// TIA Portal V17 export
// export: Created 2025-03-10T13:11:49.6492455Z, ExportSetting WithDefaults, DisplayName Totally Integrated Automation Portal, DisplayVersion V17 Update 8, DisplayName TIA Portal Openness, DisplayVersion V17 Update 8, DisplayName TIA Portal Version Control Interface, DisplayVersion V17, DisplayName SINAMICS Startdrive Advanced, DisplayVersion V17 SP2, DisplayName SINAMICS Startdrive G110M, G120, G120C, G120D, G120P, G115D, DisplayVersion V17 SP2, DisplayName SINAMICS Startdrive G130, G150, S120, S150, SINAMICS MV, S210, DisplayVersion V17 SP2, DisplayName STEP 7 Professional, DisplayVersion V17 Update 8, DisplayName SINUMERIK ONE STEP 7 Toolbox, DisplayVersion V17 Update 12, DisplayName SINUMERIK 840D sl STEP 7 Toolbox, DisplayVersion V17 Update 12, DisplayName STEP 7 Safety, DisplayVersion V17 Update 6, DisplayName WinCC Advanced, DisplayVersion V17 Update 8
VAR_GLOBAL   // PLC tag table "TAGS_IO_MPP_ITC_IPC_HT10"
   HT10_INS AT %I0.0 : "HT10_INPUTS";   // HT10 INPUTS
   HT10_OUTS AT %Q0.0 : "HT10_OUTPUTS";   // HT10 OUTPUTS
   MPP_INS AT %I120.0 : "MPP_INPUTS";   // MPP INPUTS
   MPP_OUT AT %Q120.0 : "MPP_OUTPUTS";   // MPP OUTPUTS
   TOUCH_PANEL_INPUT_1 AT %IB138 : Byte;   // TOUCH PANEL INPUT BYTE 1
   TOUCH_PANEL_INPUT_2 AT %IB139 : Byte;   // TOUCH PANEL INPUT BYTE 2
END_VAR
